(* IEC 61131-3 sources: SmartHomeNew/workspace/system_layer_cleanup/split_scaffold/core_kernel/watchdog_health_slice, 1 file *)

(* ---- FB_Watchdog_Shadow_Slice_DRAFT.st ---- *)
FUNCTION_BLOCK FB_Watchdog_Shadow_Slice_DRAFT
VAR_INPUT
    VI_System_Time_MS : UDINT;
    VI_Enable : BOOL;
END_VAR
VAR_OUTPUT
    VO_Shadow_Ready : BOOL;
END_VAR
VAR
    // Future target:
    // fbWatchdog : FB_Watchdog;
END_VAR

VO_Shadow_Ready := VI_Enable;

END_FUNCTION_BLOCK
